FUNCTION_BLOCK FB_EventF3
VAR_INPUT
	FB_Bacnet : FB_BACnet_DAIKIN_MasterStation_III_No_1;
END_VAR
VAR_OUTPUT
END_VAR
VAR
	fbMsg : FB_TcMessage;
	aUnits : ARRAY[1..22] OF AC_Unit_Status;
	stUnit   : AC_Unit_Status;
	i: INT;
	sMsgText: STRING;
	triggerTest : BOOL;
END_VAR
VAR RETAIN
	aPrevState : ARRAY[1..22] OF BOOL := [FALSE(*22*)];
END_VAR


//aUnits[1].bPresVal := FB_Bacnet.StartStopStatus_192.bPresVal;
//aUnits[1].sUnitName := 'F3-1 (1-00)';
aUnits[2].bPresVal := FB_Bacnet.StartStopStatus_193.bPresVal;
aUnits[2].sUnitName := 'F3-2 (1-01)';
aUnits[3].bPresVal := FB_Bacnet.StartStopStatus_194.bPresVal;
aUnits[3].sUnitName := 'F3-3 (1-02)';
aUnits[4].bPresVal := FB_Bacnet.StartStopStatus_195.bPresVal;
aUnits[4].sUnitName := 'F3-4 (1-03)';
aUnits[5].bPresVal := FB_Bacnet.StartStopStatus_196.bPresVal;
aUnits[5].sUnitName := 'F3-5 (1-04)';
aUnits[6].bPresVal := FB_Bacnet.StartStopStatus_197.bPresVal;
aUnits[6].sUnitName := 'F3-6 (1-05)';
aUnits[7].bPresVal := FB_Bacnet.StartStopStatus_198.bPresVal;
aUnits[7].sUnitName := 'F3-7 (1-06)';
aUnits[8].bPresVal := FB_Bacnet.StartStopStatus_199.bPresVal;
aUnits[8].sUnitName := 'F3-8 (1-07)';
aUnits[9].bPresVal := FB_Bacnet.StartStopStatus_200.bPresVal;
aUnits[9].sUnitName := 'F3-9 (1-08)';
aUnits[10].bPresVal := FB_Bacnet.StartStopStatus_201.bPresVal;
aUnits[10].sUnitName := 'F3-10 (1-09)';
aUnits[11].bPresVal := FB_Bacnet.StartStopStatus_202.bPresVal;
aUnits[11].sUnitName := 'F3-11 (1-10)';
aUnits[12].bPresVal := FB_Bacnet.StartStopStatus_203.bPresVal;
aUnits[12].sUnitName := 'F3-12 (1-11)';
aUnits[13].bPresVal := FB_Bacnet.StartStopStatus_204.bPresVal;
aUnits[13].sUnitName := 'F3-13 (1-12)';
aUnits[14].bPresVal := FB_Bacnet.StartStopStatus_205.bPresVal;
aUnits[14].sUnitName := 'F3-14 (1-13)';
aUnits[15].bPresVal := FB_Bacnet.StartStopStatus_206.bPresVal;
aUnits[15].sUnitName := 'F3-15 (1-14)';
aUnits[16].bPresVal := FB_Bacnet.StartStopStatus_207.bPresVal;
aUnits[16].sUnitName := 'F3-16 (1-15)';
aUnits[17].bPresVal := FB_Bacnet.StartStopStatus_208.bPresVal;
aUnits[17].sUnitName := 'F3-17 (2-00)';
aUnits[18].bPresVal := FB_Bacnet.StartStopStatus_209.bPresVal;
aUnits[18].sUnitName := 'F3-18 (2-01)';
aUnits[19].bPresVal := FB_Bacnet.StartStopStatus_210.bPresVal;
aUnits[19].sUnitName := 'F3-19 (2-02)';
aUnits[20].bPresVal := FB_Bacnet.StartStopStatus_211.bPresVal;
aUnits[20].sUnitName := 'F3-20 (2-03)';
aUnits[21].bPresVal := FB_Bacnet.StartStopStatus_212.bPresVal;
aUnits[21].sUnitName := 'F3-21 (2-04)';
aUnits[22].bPresVal := FB_Bacnet.StartStopStatus_224.bPresVal;
aUnits[22].sUnitName := 'F3-Lobi (3-00)';

FOR i := 1 TO 22 DO
	stUnit := aUnits[i]; // extract the structure instance
    IF aUnits[i].bPresVal <> aPrevState[i] THEN
        IF aUnits[i].bPresVal THEN
            sMsgText := CONCAT(stUnit.sUnitName, ' is Turned ON');
        ELSE
            sMsgText := CONCAT(stUnit.sUnitName, ' is Turned OFF');
        END_IF
		fbMsg.CreateEx(TC_EVENTS.UnitPowerStatus.EventPowerStatus, 0);
		fbMsg.ipArguments.AddString(sMsgText);
		fbMsg.Send(0);
		
        // Update previous state
        aPrevState[i] := aUnits[i].bPresVal;
    END_IF
END_FOR

END_FUNCTION_BLOCK

(* stored: Version 1.1.0.1, ProductVersion 3.1.4024.14
   POU FB_EventF3: Id {6aa3eb25-9366-4388-b87e-cc7a1459f595}, SpecialFunc None *)
